// TIA Portal V19 export
DATA_BLOCK "A0302_PERS"   // DB107
// stored: MemoryReserve 100
   VAR RETAIN
      Par : Struct
         CarroPareggCoda : Struct
            Delay_StartMove : Time;
            Preset { S7_SetPoint := 'True'} : LReal := 435.433;
         END_STRUCT;
         CarroPareggTesta : Struct
            Delay_StartMove : Time;
            Preset { S7_SetPoint := 'True'} : LReal := 348.633;
         END_STRUCT;
         Cremaliera : Struct
            Modulo { S7_SetPoint := 'True'} : LReal := 2.5;
            Passo { S7_SetPoint := 'True'} : LReal := 7.854;
         END_STRUCT;
      END_STRUCT;
   END_VAR
BEGIN
END_DATA_BLOCK
